// TIA Portal V18 export
TYPE "AHUChannel_v1"
// stored: IsFailsafeCompliant false
   STRUCT
      SAFCmd1 : Array[0..2] of Bool;
      SAFCmd2 : Array[0..2] of Bool;
      SAFCmd3 : Array[0..2] of Bool;
      SAFSpeed1Ind : Array[0..2] of Bool;   // Off/On
      SAFSpeed2Ind : Array[0..2] of Bool;   // Off/On
      SAFIsBlockedByFrostProt : Array[0..2] of Bool;   // Off/On
      SAFInd4 : Array[0..2] of Bool;
      SAFInd5 : Array[0..2] of Bool;
      SAFInd6 : Array[0..2] of Bool;
      SAFInd7 : Array[0..2] of Bool;
      HeaterRlyIsOn : Array[0..2] of Bool;   // Off/On
      HeaterRlyIsOff : Array[0..2] of Bool;   // Off/On
      HeaterRlyOnCmd : Array[0..2] of Bool;   // Off/On
      HeaterInitialSignal : Array[0..2] of Real;   // 0-100.0%
      HeaterAdaptedSignal : Array[0..2] of Real;   // 0-100.0%
      MixingRlyIsOn : Array[0..2] of Bool;   // Off/On
      MixingRlyIsOff : Array[0..2] of Bool;   // Off/On
      MixingRlyOnCmd : Array[0..2] of Bool;   // Off/On
      MixingInitialSignal : Array[0..2] of Real;   // 0-100.0%
      MixingAdaptedSignal : Array[0..2] of Real;   // 0-100.0%
      ExtractRlyIsOn : Array[0..2] of Bool;   // Off/On
      ExtractRlyIsOff : Array[0..2] of Bool;   // Off/On
      ExtractRlyOnCmd : Array[0..2] of Bool;   // Off/On
      ExtractInitialSignal : Array[0..2] of Real;   // 0-100.0%
      ExtractAdaptedSignal : Array[0..2] of Real;   // 0-100.0%
   END_STRUCT;
END_TYPE
